(* Logix 5000 project; controller CLASE_1 Emulate 5570 rev 28.11; software revision 28.02; part 15 of 15 *)
(* tags used below, declared in another part *)
   COCCION_TK_200 : TIMER;
   Cond1_Nivel_TK_200 : BOOL;
   Cond2_Nivel_TK_200 : BOOL;
   Cond3_Nivel_TK_200 : BOOL;
   E0_Calentar_TK_200 : SFC_STEP;
   E0_Llenar_TK_100 : SFC_STEP;
   E0_Llenar_TK_200 : SFC_STEP;
   E0_Moler_TK_300 : SFC_STEP;
   E0_Vaciado_TK_300 : SFC_STEP;
   E1_Calentar_TK_200 : SFC_STEP;
   E1_LLenar_TK_100 : SFC_STEP;
   E1_LLenar_TK_200 : SFC_STEP;
   E1_LLenar_TK_300 : SFC_STEP;
   E1_Vaciado_TK_300 : SFC_STEP;
   E2_Agitar_TK_200 : SFC_STEP;
   E2_Trirurado_TK_100 : SFC_STEP;
   E3_Calentar_TK_300 : SFC_STEP;
   E4_Moler_TK_300 : SFC_STEP;
   FV_100 : P_ValveSO;
   FV_100_Intlk : P_Intlk;
   FV_100_Perm : P_Perm;
   LIT_200 : P_AIn;
   Llenar_T2 : BOOL;
   Llenar_TK_100 : BOOL;
   LSH_100 : P_DIn;
   M_100 : P_VSD;
   M_200 : P_VSD;
   M_300 : P_VSD;
   Nivel_TK_200 : BOOL;
   P_100_B : P_VSD;
   P_200 : P_VSD;
   P_300 : P_VSD;
   PID_Auto_mode : BOOL;
   PID_OUT_TK_200 : REAL;   // Esfuerzo de control Deberá ir direccionada a la salida analogica fisica
   PID_OUT_TK_300 : REAL;
   PID_TT : PIDE_AUTOTUNE;
   PID_TT3 : PIDE_AUTOTUNE;
   Pump_100_A : P_VSD;
   SET_POINT_2_Temperatura : REAL;
   SET_POINT_3_Temperatura : REAL;
   SP_Timer_M_100 : TIMER;
   Sp_Timer_P_200 : TIMER;
   SP_Timer_P_300 : TIMER;
   Sp_veloc_M_200 : DINT;
   SP_veloc_P_100_B : DINT;
   SP_veloc_Pump_100_A : DINT;
   Temperatura_ok : BOOL;
   Temperatura_TT_200 : REAL;
   Temperatura_TT_300 : REAL;
   Timer_molienda_ctrlTemp : TIMER;

PROGRAM MainProgram   (* main routine MainRoutine *)

ROUTINE MainRoutine   (* ladder *)
END_ROUTINE
END_PROGRAM

PROGRAM PID_Controllers   (* main routine Main *)
VAR
   BNOT_01 : FBD_BOOLEAN_NOT := (In := 1);
   BNOT_02 : FBD_BOOLEAN_NOT := (In := 1);
   BNOT_03 : FBD_BOOLEAN_NOT := (In := 1);
   P_FT_Primer_Orden_AOI_01 : P_FT_Primer_Orden_AOI := (Kp := 1.0, Tao := 5.0, Inp_Sistema := 59.999977, Out_Sistema := 59.99998, Tiempo_muerto := 1.5, FT_EnableIN := 1);
   P_FT_Primer_Orden_AOI_02 : P_FT_Primer_Orden_AOI := (Kp := 1.0, Tao := 5.0, Out_Sistema := 59.99998, Tiempo_muerto := 1.5, FT_EnableIN := 1);
   P_FT_Primer_Orden_AOI_03 : P_FT_Primer_Orden_AOI := (Kp := 1.0, Tao := 5.0, Inp_Sistema := 59.999977, Out_Sistema := 59.99998, Tiempo_muerto := 1.5, FT_EnableIN := 1);
   PIDE_01 : PID_ENHANCED := (PV := 59.99998, PVEUMax := 100.0, SPProg := 60.0, SPOper := 60.0, SPHLimit := 100.0, RatioProg := 1.0, RatioOper := 1.0, RatioHLimit := 1.0, RatioLLimit := 1.0, CVOper := 59.999977, CVEUMax := 100.0, CVHLimit := 100.0, PGain := 1.8545046, IGain := 18.341255, DGain := 0.020605609, PVEDerivative := 1, ProgProgReq := 1, ProgAutoReq := 1, RTSTime := 1, CVEU := 59.999977, CV := 59.999977, SP := 60.0, SPPercent := 60.0, PVPercent := 59.99998, E := 1.9073486e-05, EPercent := 1.9073486e-05, InitPrimary := 1, Ratio := 1.0, ProgOper := 1, Auto := 1, DeltaT := 0.2, AtuneReady := 1, AtuneDone := 1);
   PIDE_02 : PID_ENHANCED := (PV := 59.99998, PVEUMax := 200.0, SPProg := 60.0, SPOper := 60.0, SPHLimit := 200.0, RatioProg := 1.0, RatioOper := 1.0, RatioHLimit := 1.0, RatioLLimit := 1.0, CVOper := 59.999977, CVEUMax := 200.0, CVHLimit := 100.0, PGain := 1.8545046, IGain := 18.341255, DGain := 0.020605609, PVEDerivative := 1, ProgProgReq := 1, ProgAutoReq := 1, RTSTime := 1, CVEU := 59.999977, CV := 59.999977, SP := 60.0, SPPercent := 60.0, PVPercent := 59.99998, E := 1.9073486e-05, EPercent := 1.9073486e-05, InitPrimary := 1, Ratio := 1.0, ProgOper := 1, Auto := 1, DeltaT := 0.2, AtuneReady := 1, AtuneDone := 1);
   PIDE_03 : PID_ENHANCED := (PV := 59.99998, PVEUMax := 100.0, SPProg := 60.0, SPOper := 60.0, SPHLimit := 100.0, RatioProg := 1.0, RatioOper := 1.0, RatioHLimit := 1.0, RatioLLimit := 1.0, CVOper := 59.999977, CVEUMax := 100.0, CVHLimit := 100.0, PGain := 1.8545046, IGain := 18.341255, DGain := 0.020605609, PVEDerivative := 1, ProgProgReq := 1, ProgAutoReq := 1, RTSTime := 1, CVEU := 59.999977, CV := 59.999977, SP := 60.0, SPPercent := 60.0, PVPercent := 59.99998, E := 1.9073486e-05, EPercent := 1.9073486e-05, InitPrimary := 1, Ratio := 1.0, ProgOper := 1, Auto := 1, DeltaT := 0.2, AtuneReady := 1, AtuneDone := 1);
END_VAR

ROUTINE _00_FT_Primer_Orden   (* function block diagram *)
   SHEET 1   // FT_TK_200
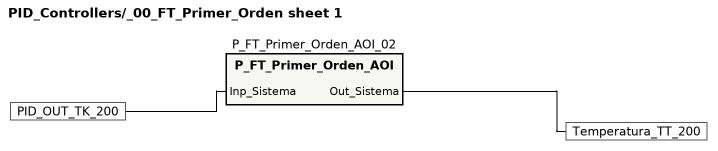
   P_FT_Primer_Orden_AOI_02 : P_FT_Primer_Orden_AOI(Inp_Sistema := PID_OUT_TK_200);
   Temperatura_TT_200 := P_FT_Primer_Orden_AOI_02.Out_Sistema;
   SHEET 2   // FT_TK_300
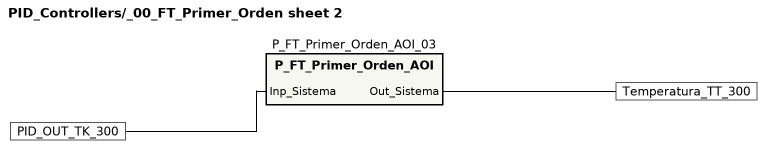
   P_FT_Primer_Orden_AOI_03 : P_FT_Primer_Orden_AOI(Inp_Sistema := PID_OUT_TK_300);
   Temperatura_TT_300 := P_FT_Primer_Orden_AOI_03.Out_Sistema;
END_ROUTINE

ROUTINE _01_PIDs   (* function block diagram *)
   SHEET 1   // PID_TK_200
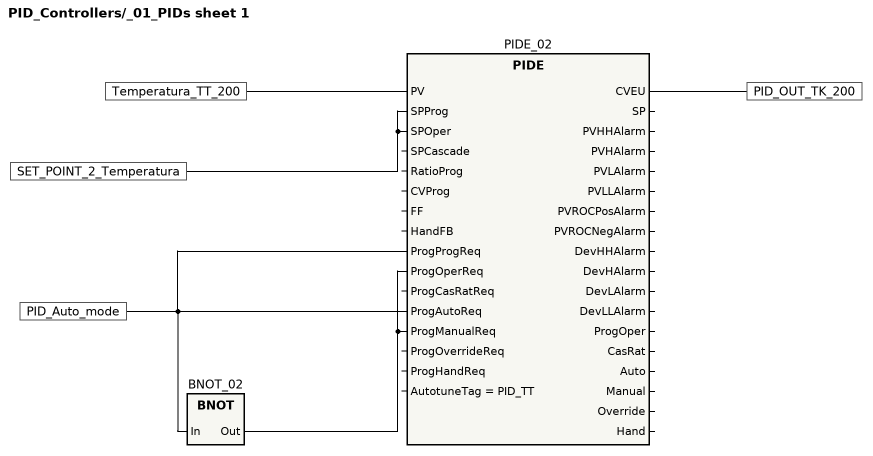
   BNOT_02 : BNOT(In := PID_Auto_mode);
   PIDE_02 : PIDE(PV := Temperatura_TT_200, SPProg := SET_POINT_2_Temperatura, SPOper := SET_POINT_2_Temperatura, ProgProgReq := PID_Auto_mode, ProgOperReq := BNOT_02.Out, ProgAutoReq := PID_Auto_mode, ProgManualReq := BNOT_02.Out, AutotuneTag := PID_TT);   // unwired pins: SPCascade RatioProg CVProg FF HandFB ProgCasRatReq ProgOverrideReq ProgHandReq SP PVHHAlarm PVHAlarm PVLAlarm PVLLAlarm PVROCPosAlarm PVROCNegAlarm DevHHAlarm DevHAlarm DevLAlarm DevLLAlarm ProgOper CasRat Auto Manual Override Hand
   PID_OUT_TK_200 := PIDE_02.CVEU;
   SHEET 2   // PID_TK_300
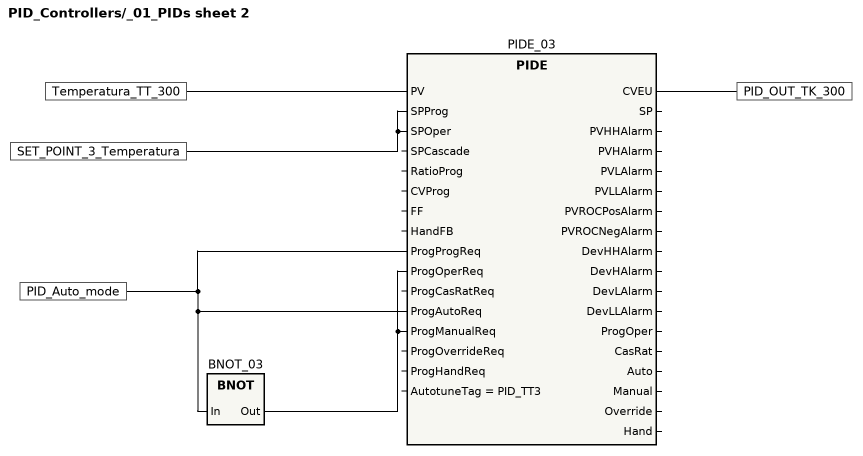
   BNOT_03 : BNOT(In := PID_Auto_mode);
   PIDE_03 : PIDE(PV := Temperatura_TT_300, SPProg := SET_POINT_3_Temperatura, SPOper := SET_POINT_3_Temperatura, ProgProgReq := PID_Auto_mode, ProgOperReq := BNOT_03.Out, ProgAutoReq := PID_Auto_mode, ProgManualReq := BNOT_03.Out, AutotuneTag := PID_TT3);   // unwired pins: SPCascade RatioProg CVProg FF HandFB ProgCasRatReq ProgOverrideReq ProgHandReq SP PVHHAlarm PVHAlarm PVLAlarm PVLLAlarm PVROCPosAlarm PVROCNegAlarm DevHHAlarm DevHAlarm DevLAlarm DevLLAlarm ProgOper CasRat Auto Manual Override Hand
   PID_OUT_TK_300 := PIDE_03.CVEU;
END_ROUTINE

ROUTINE Main   (* ladder *)
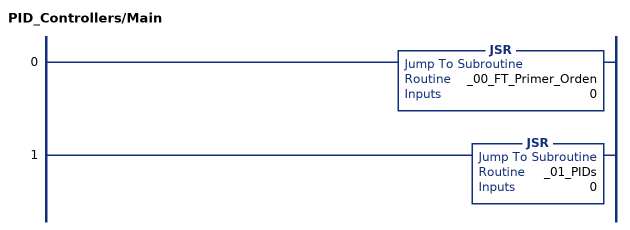
   0: JSR(_00_FT_Primer_Orden,0);
   1: JSR(_01_PIDs,0);
END_ROUTINE
END_PROGRAM

PROGRAM SEC_Proceso_Chocolate_SFC   (* main routine Main *)
VAR
   Action_000 : SFC_ACTION := (Status := 16#0020_0000, PauseTimer := 1);
   Action_001 : SFC_ACTION := (Status := 16#0020_0000, PauseTimer := 1);
   Action_002 : SFC_ACTION := (Status := 16#c020_0000, A := 1, Q := 1, PauseTimer := 1, Count := 1);
   Action_003 : SFC_ACTION := (Status := 16#0020_0000, PauseTimer := 1);
   Action_004 : SFC_ACTION := (Status := 16#0020_0000, PauseTimer := 1);
   Action_005 : SFC_ACTION := (Status := 16#0020_0000, PauseTimer := 1);
   Action_006 : SFC_ACTION := (Status := 16#0020_0000, PauseTimer := 1);
   Action_007 : SFC_ACTION := (Status := 16#0020_0000, PauseTimer := 1);
   Action_008 : SFC_ACTION := (Status := 16#0020_0000, PauseTimer := 1);
   Action_009 : SFC_ACTION := (Status := 16#0020_0000, PauseTimer := 1);
   Action_010 : SFC_ACTION := (Status := 16#0020_0000, PauseTimer := 1);
   Action_011 : SFC_ACTION := (Status := 16#0020_0000, PauseTimer := 1);
   Action_012 : SFC_ACTION := (Status := 16#0020_0000, PauseTimer := 1);
   Action_013 : SFC_ACTION := (Status := 16#0020_0000, PauseTimer := 1);
   P_DIn_01 : P_DIn := (Inp_PV := 1, Inp_Target := 1, Inp_Gate := 1, Cfg_NormTextVis := 1, Cfg_PCmdClear := 1, Cfg_TgtDisagreeAckReqd := 1, Cfg_TgtDisagreeSeverity := 750, Ack_TgtDisagree := 1);
   P_ValveSO_01 : P_ValveSO := (Inp_PermOK := 1, Inp_NBPermOK := 1, Inp_IntlkOK := 1, Inp_NBIntlkOK := 1, Cfg_LSFail := 1, Cfg_PCmdClear := 1, Cfg_ProgDefault := 1, Cfg_ShedOnFullStall := 1, Cfg_ShedOnTransitStall := 1, Cfg_ShedOnIOFault := 1, Cfg_FullStallAckReqd := 1, Cfg_TransitStallAckReqd := 1, Cfg_IntlkTripAckReqd := 1, Cfg_IOFaultAckReqd := 1, Cfg_FullStallSeverity := 1000, Cfg_TransitStallSeverity := 1000, Cfg_IntlkTripSeverity := 500, Cfg_IOFaultSeverity := 1000, Cfg_SimFdbkT := 2, Cfg_FullStallT := 5, Cfg_TransitStallT := 10, Ack_FullStall := 1, Ack_TransitStall := 1, Ack_IntlkTrip := 1, Ack_IOFault := 1);
   Step_000 : SFC_STEP := (Status := 16#0020_0000, PauseTimer := 1);
   Step_001 : SFC_STEP := (Status := 16#0020_0000, PauseTimer := 1);
   Step_002 : SFC_STEP := (Status := 16#0020_0000, PauseTimer := 1);
   Step_003 : SFC_STEP := (Status := 16#0020_0000, PauseTimer := 1);
   Step_004 : SFC_STEP := (Status := 16#0020_0000, PauseTimer := 1);
   Step_005 : SFC_STEP := (Status := 16#0020_0000, PauseTimer := 1);
   Step_006 : SFC_STEP := (Status := 16#0020_0000, PauseTimer := 1);
   Step_007 : SFC_STEP := (Status := 16#0020_0000, PauseTimer := 1);
   Step_008 : SFC_STEP := (Status := 16#0020_0000, PauseTimer := 1);
   Step_009 : SFC_STEP := (Status := 16#0020_0000, PauseTimer := 1);
   Step_010 : SFC_STEP := (Status := 16#0020_0000, PauseTimer := 1);
   Step_011 : SFC_STEP := (Status := 16#0020_0000, PauseTimer := 1);
   Step_012 : SFC_STEP := (Status := 16#0020_0000, PauseTimer := 1);
   Step_013 : SFC_STEP := (Status := 16#0020_0000, PauseTimer := 1);
   Step_014 : SFC_STEP := (Status := 16#0020_0000, PauseTimer := 1);
   Step_015 : SFC_STEP := (Status := 16#0020_0000, PauseTimer := 1);
   Step_016 : SFC_STEP := (Status := 16#0020_0000, PauseTimer := 1);
   Step_017 : SFC_STEP := (Status := 16#0020_0000, PauseTimer := 1);
   Step_018 : SFC_STEP := (Status := 16#0020_0000, PauseTimer := 1);
   Step_019 : SFC_STEP := (Status := 16#0020_0000, PauseTimer := 1);
   Step_020 : SFC_STEP := (Status := 16#0020_0000, PauseTimer := 1);
   Step_021 : SFC_STEP := (Status := 16#0020_0000, PauseTimer := 1);
   Step_022 : SFC_STEP := (Status := 16#0020_0000, PauseTimer := 1);
   Tran_000 : BOOL;
   Tran_001 : BOOL;
   Tran_002 : BOOL;
   Tran_003 : BOOL;
   Tran_004 : BOOL;
   Tran_005 : BOOL;
   Tran_006 : BOOL;
   Tran_007 : BOOL;
   Tran_008 : BOOL;
   Tran_009 : BOOL;
   Tran_010 : BOOL;
   Tran_011 : BOOL;
   Tran_012 : BOOL;
   Tran_013 : BOOL;
   Tran_014 : BOOL;
END_VAR

ROUTINE Acciones   (* ladder *)
// Es lo que tiene que ver con etapas
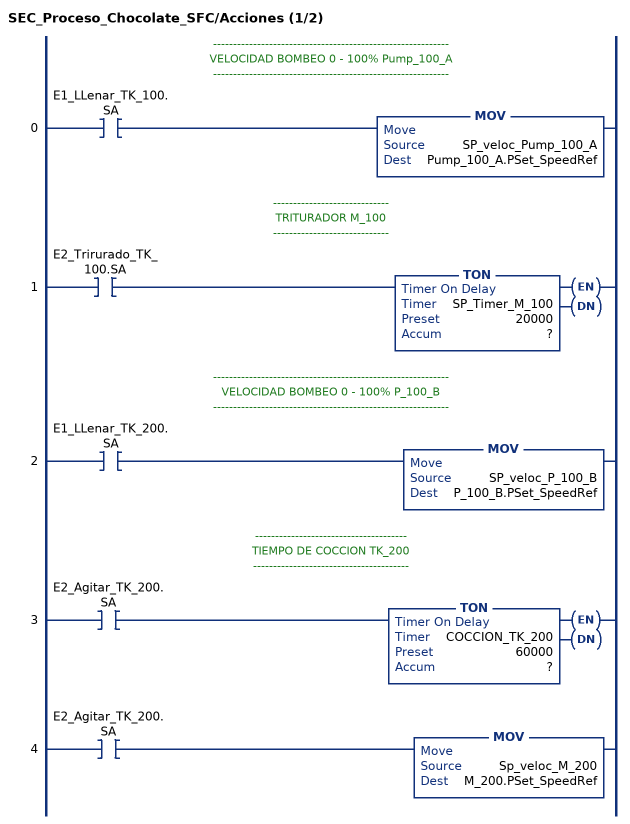
   // -----------------------------------------------------------
   // VELOCIDAD BOMBEO 0 - 100% Pump_100_A
   // -----------------------------------------------------------
   0: XIC(E1_LLenar_TK_100.SA)MOV(SP_veloc_Pump_100_A,Pump_100_A.PSet_SpeedRef);
   // -----------------------------
   // TRITURADOR M_100
   // -----------------------------
   1: XIC(E2_Trirurado_TK_100.SA)TON(SP_Timer_M_100,?,?);
   // -----------------------------------------------------------
   // VELOCIDAD BOMBEO 0 - 100% P_100_B
   // -----------------------------------------------------------
   2: XIC(E1_LLenar_TK_200.SA)MOV(SP_veloc_P_100_B,P_100_B.PSet_SpeedRef);
   // --------------------------------------
   // TIEMPO DE COCCION TK_200
   // ---------------------------------------
   3: XIC(E2_Agitar_TK_200.SA)TON(COCCION_TK_200,?,?);
   4: XIC(E2_Agitar_TK_200.SA)MOV(Sp_veloc_M_200,M_200.PSet_SpeedRef);
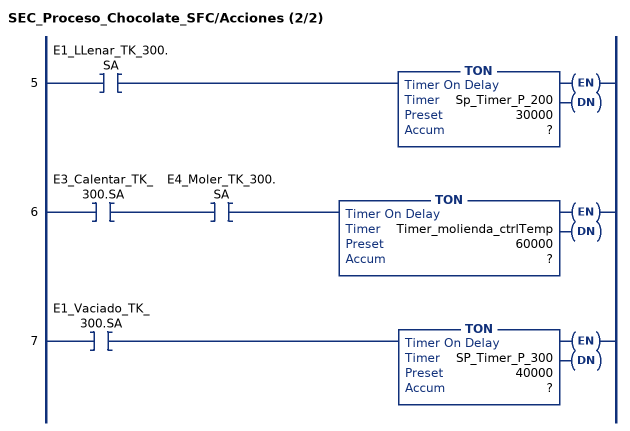
   5: XIC(E1_LLenar_TK_300.SA)TON(Sp_Timer_P_200,?,?);
   6: XIC(E3_Calentar_TK_300.SA)XIC(E4_Moler_TK_300.SA)TON(Timer_molienda_ctrlTemp,?,?);
   7: XIC(E1_Vaciado_TK_300.SA)TON(SP_Timer_P_300,?,?);
END_ROUTINE

ROUTINE Condiciones   (* ladder *)
// Es lo que tiene que ver con transiciones
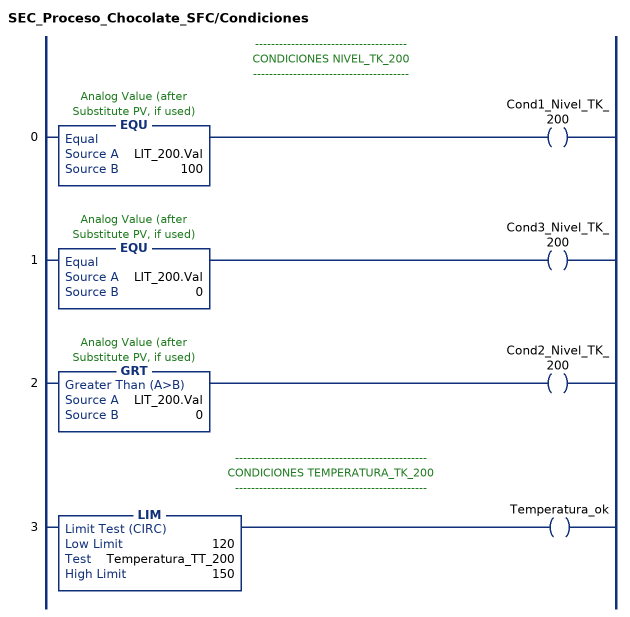
   // --------------------------------------
   // CONDICIONES NIVEL_TK_200
   // ---------------------------------------
   0: EQU(LIT_200.Val,100)OTE(Cond1_Nivel_TK_200);
   1: EQU(LIT_200.Val,0)OTE(Cond3_Nivel_TK_200);
   2: GRT(LIT_200.Val,0)OTE(Cond2_Nivel_TK_200);
   // ------------------------------------------------
   // CONDICIONES TEMPERATURA_TK_200
   // ------------------------------------------------
   3: LIM(120,Temperatura_TT_200,150)OTE(Temperatura_ok);
END_ROUTINE

ROUTINE Main   (* ladder *)
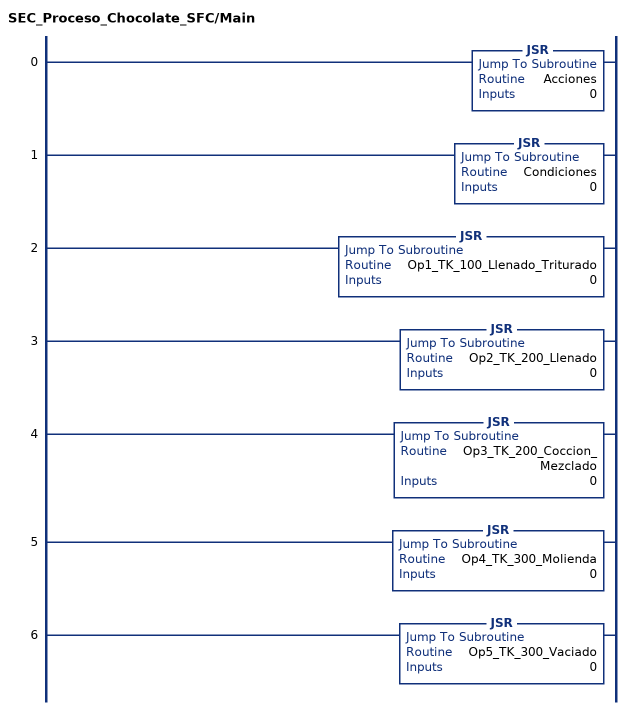
   0: JSR(Acciones,0);
   1: JSR(Condiciones,0);
   2: JSR(Op1_TK_100_Llenado_Triturado,0);
   3: JSR(Op2_TK_200_Llenado,0);
   4: JSR(Op3_TK_200_Coccion_Mezclado,0);
   5: JSR(Op4_TK_300_Molienda,0);
   6: JSR(Op5_TK_300_Vaciado,0);
END_ROUTINE

ROUTINE Op1_TK_100_Llenado_Triturado   (* sequential function chart *)
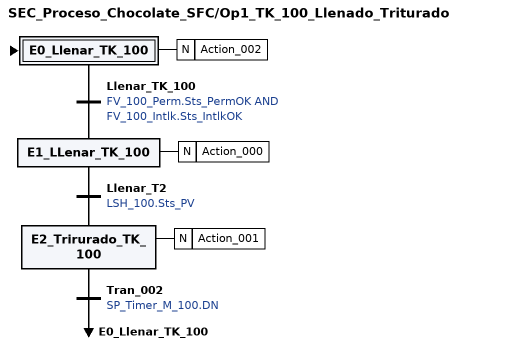
   INITIAL_STEP E0_Llenar_TK_100:
      ACTION Action_002 (N):
         //RESET DE EQUIPOS
         FV_100.PCmd_Close:= 1;
         Pump_100_A.PCmd_Stop:=1;
         Pump_100_A.PSet_SpeedRef:=0;
         M_100.PCmd_Stop:=1;
         
      END_ACTION
   END_STEP
   TRANSITION Llenar_TK_100 FROM E0_Llenar_TK_100 TO E1_LLenar_TK_100
      := FV_100_Perm.Sts_PermOK AND FV_100_Intlk.Sts_IntlkOK
   END_TRANSITION
   STEP E1_LLenar_TK_100:
      ACTION Action_000 (N):
         // Activar equipos de llenado
         FV_100.PCmd_Open:= 1;
      END_ACTION
   END_STEP
   TRANSITION Llenar_T2 FROM E1_LLenar_TK_100 TO E2_Trirurado_TK_100
      := LSH_100.Sts_PV
   END_TRANSITION
   STEP E2_Trirurado_TK_100:
      ACTION Action_001 (N):
         M_100.PCmd_Start:=1;
         FV_100.PCmd_Close:= 1;
         Pump_100_A.PCmd_Start:= 1;
      END_ACTION
   END_STEP
   TRANSITION Tran_002 FROM E2_Trirurado_TK_100 TO E0_Llenar_TK_100
      := SP_Timer_M_100.DN
   END_TRANSITION
END_ROUTINE

ROUTINE Op2_TK_200_Llenado   (* sequential function chart *)
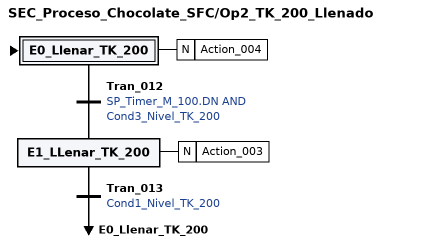
   INITIAL_STEP E0_Llenar_TK_200:
      ACTION Action_004 (N):
         //RESET DE EQUIPOS
         P_100_B.PCmd_Stop:= 1;
         P_100_B.PSet_SpeedRef:=0;
         
      END_ACTION
   END_STEP
   TRANSITION Tran_012 FROM E0_Llenar_TK_200 TO E1_LLenar_TK_200
      :=  SP_Timer_M_100.DN AND Cond3_Nivel_TK_200
   END_TRANSITION
   STEP E1_LLenar_TK_200:
      ACTION Action_003 (N):
         P_100_B.PCmd_Start:= 1;
      END_ACTION
   END_STEP
   TRANSITION Tran_013 FROM E1_LLenar_TK_200 TO E0_Llenar_TK_200
      := Cond1_Nivel_TK_200
   END_TRANSITION
END_ROUTINE

ROUTINE Op3_TK_200_Coccion_Mezclado   (* sequential function chart *)
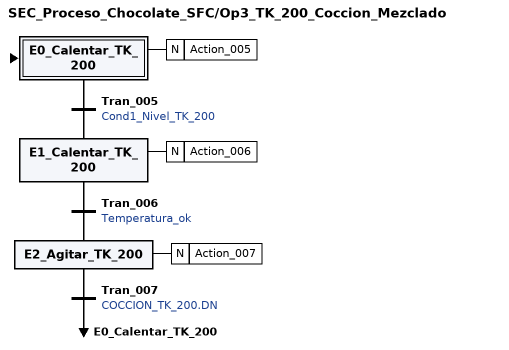
   INITIAL_STEP E0_Calentar_TK_200:
      ACTION Action_005 (N):
         //RESET DE EQUIPOS
         SET_POINT_2_Temperatura:=0;
         M_200.PCmd_Stop:=1;
         M_200.PSet_SpeedRef:=0;
      END_ACTION
   END_STEP
   TRANSITION Tran_005 FROM E0_Calentar_TK_200 TO E1_Calentar_TK_200
      := Cond1_Nivel_TK_200
   END_TRANSITION
   STEP E1_Calentar_TK_200:
      ACTION Action_006 (N):
         SET_POINT_2_Temperatura:=135;
         P_100_B.PCmd_Stop:=1;
         P_100_B.PSet_SpeedRef:=0;
      END_ACTION
   END_STEP
   TRANSITION Tran_006 FROM E1_Calentar_TK_200 TO E2_Agitar_TK_200
      := Temperatura_ok
   END_TRANSITION
   STEP E2_Agitar_TK_200:
      ACTION Action_007 (N):
         M_200.PCmd_Start:=1;
      END_ACTION
   END_STEP
   TRANSITION Tran_007 FROM E2_Agitar_TK_200 TO E0_Calentar_TK_200
      := COCCION_TK_200.DN
   END_TRANSITION
END_ROUTINE

ROUTINE Op4_TK_300_Molienda   (* sequential function chart *)
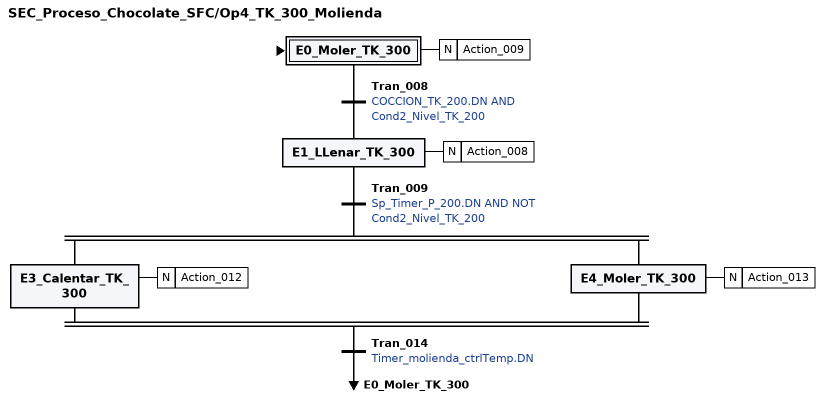
   INITIAL_STEP E0_Moler_TK_300:
      ACTION Action_009 (N):
         //RESET DE EQUIPOS
         P_200.PCmd_Stop:=1;
         SET_POINT_3_Temperatura:=0;
         M_300.PCmd_Stop:=1;
      END_ACTION
   END_STEP
   TRANSITION Tran_008 FROM E0_Moler_TK_300 TO E1_LLenar_TK_300
      := COCCION_TK_200.DN AND Cond2_Nivel_TK_200
   END_TRANSITION
   STEP E1_LLenar_TK_300:
      ACTION Action_008 (N):
         P_200.PCmd_Start:=1;
      END_ACTION
   END_STEP
   TRANSITION Tran_009 FROM E1_LLenar_TK_300 TO (E4_Moler_TK_300, E3_Calentar_TK_300)
      := Sp_Timer_P_200.DN AND NOT Cond2_Nivel_TK_200
   END_TRANSITION
   STEP E3_Calentar_TK_300:
      ACTION Action_012 (N):
         SET_POINT_3_Temperatura:=75;
      END_ACTION
   END_STEP
   STEP E4_Moler_TK_300:
      ACTION Action_013 (N):
         M_300.PCmd_Start:=1;
      END_ACTION
   END_STEP
   TRANSITION Tran_014 FROM (E3_Calentar_TK_300, E4_Moler_TK_300) TO E0_Moler_TK_300
      := Timer_molienda_ctrlTemp.DN
   END_TRANSITION
END_ROUTINE

ROUTINE Op5_TK_300_Vaciado   (* sequential function chart *)
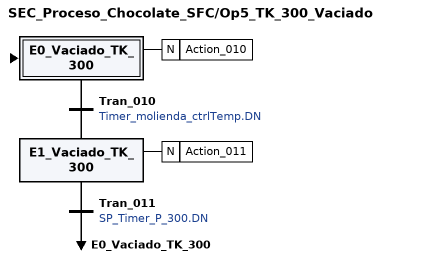
   INITIAL_STEP E0_Vaciado_TK_300:
      ACTION Action_010 (N):
         P_300.PCmd_Stop:=1;
      END_ACTION
   END_STEP
   TRANSITION Tran_010 FROM E0_Vaciado_TK_300 TO E1_Vaciado_TK_300
      := Timer_molienda_ctrlTemp.DN
   END_TRANSITION
   STEP E1_Vaciado_TK_300:
      ACTION Action_011 (N):
         P_300.PCmd_Start:=1;
      END_ACTION
   END_STEP
   TRANSITION Tran_011 FROM E1_Vaciado_TK_300 TO E0_Vaciado_TK_300
      := SP_Timer_P_300.DN
   END_TRANSITION
END_ROUTINE
END_PROGRAM
